(* IEC 61131-3 sources: Lasal/CPU_5344_V01/Class/switchesAxis, 1 file *)

(* ---- switchesAxis.st ---- *)
(*!
<Class
	Name               = "switchesAxis"
	Revision           = "0.0"
	RealtimeTask       = "false"
	CyclicTask         = "false"
	BackgroundTask     = "false"
	Sigmatek           = "false"
	OSInterface        = "false"
	HighPriority       = "false"
	Automatic          = "false"
	UpdateMode         = "Prescan"
	SharedCommandTable = "true"
	Objectsize         = "(284,120)">
	<Channels>
		<Server Name="ClassSvr" Visualized="false" Initialize="false" WriteProtected="true" Retentive="false"/>
		<Server Name="maxSwitch" Visualized="false" Initialize="false" WriteProtected="true" Retentive="false"/>
		<Server Name="minSwitch" Visualized="false" Initialize="false" WriteProtected="true" Retentive="false"/>
		<Server Name="overRuleMax" Visualized="false" Initialize="false" WriteProtected="false" Retentive="false"/>
		<Server Name="overRuleMin" Visualized="false" Initialize="false" WriteProtected="false" Retentive="false"/>
		<Server Name="overRuleRef" Visualized="false" Initialize="false" WriteProtected="false" Retentive="false"/>
		<Server Name="refSwitch" Visualized="false" Initialize="false" WriteProtected="true" Retentive="false"/>
		<Server Name="switchMaxIsNormallyOpen" Visualized="false" Initialize="false" WriteProtected="false" Retentive="File"/>
		<Server Name="switchMinIsNormallyOpen" Visualized="false" Initialize="false" WriteProtected="false" Retentive="File"/>
		<Client Name="ctrlServo" Required="true" Internal="false"/>
		<Client Name="iEsMaxSwitch" Required="false" Internal="false"/>
		<Client Name="iEsMinSwitch" Required="false" Internal="false"/>
		<Client Name="iEsRefSwitch" Required="false" Internal="false"/>
	</Channels>
</Class>
*)
switchesAxis : CLASS
  //Servers:
	ClassSvr 	: SvrChCmd_DINT;
	minSwitch 	: SvrCh_DINT;
	maxSwitch 	: SvrCh_DINT;
	refSwitch 	: SvrCh_DINT;
	switchMinIsNormallyOpen 	: SvrCh_DINT;
	switchMaxIsNormallyOpen 	: SvrCh_DINT;
	overRuleMin 	: SvrCh_DINT;
	overRuleMax 	: SvrCh_DINT;
	overRuleRef 	: SvrCh_DINT;
  //Clients:
	iEsMinSwitch 	: CltCh_DINT;
	iEsMaxSwitch 	: CltCh_DINT;
	iEsRefSwitch 	: CltCh_DINT;
	ctrlServo 	: CltChCmd_cmServo;
  //Variables:
  //Functions:

	FUNCTION VIRTUAL GLOBAL minSwitch::Read
		VAR_OUTPUT
			output (EAX) 	: DINT;
		END_VAR;

	FUNCTION VIRTUAL GLOBAL maxSwitch::Read
		VAR_OUTPUT
			output (EAX) 	: DINT;
		END_VAR;

	FUNCTION VIRTUAL GLOBAL refSwitch::Read
		VAR_OUTPUT
			output (EAX) 	: DINT;
		END_VAR;
  //Tables:
	FUNCTION @STD
		VAR_OUTPUT
			ret_code	: CONFSTATES;
		END_VAR;
	FUNCTION GLOBAL TAB @CT_;
END_CLASS;

#pragma usingLtd cmServo

// JdK 22-3-2022: switchesAxis, connect the endswitches to the axis, also handles the simulation states, goal is to make it less work to go to and from simulation

FUNCTION VIRTUAL GLOBAL switchesAxis::minSwitch::Read
	VAR_OUTPUT
		output (EAX) 	: DINT;
	END_VAR

  iEsMinSwitch:= iEsMinSwitch.Read();
  IF overRuleMin<> 0 THEN
   minSwitch:= overRuleMin>0;
  ELSIF ctrlServo.stsAllSimuActive THEN
    IF ctrlServo.parRefDirPositive= 0 THEN
      minSwitch:= ctrlServo.stsSimRef; //homing negative
    ELSE
      minSwitch:= 0;
    END_IF;
  ELSE
    IF switchMinIsNormallyOpen THEN
      minSwitch:= iEsMinSwitch;
    ELSE
      minSwitch:= iEsMinSwitch= 0; //invert signal
    END_IF;
  END_IF;

	output := minSwitch;

END_FUNCTION

FUNCTION VIRTUAL GLOBAL switchesAxis::maxSwitch::Read
	VAR_OUTPUT
		output (EAX) 	: DINT;
	END_VAR

  iEsMaxSwitch:= iEsMaxSwitch.Read();
  IF overRuleMax<> 0 THEN
    maxSwitch:= overRuleMax>0;
  ELSIF ctrlServo.stsAllSimuActive THEN
    IF ctrlServo.parRefDirPositive= 1 THEN
      maxSwitch:= ctrlServo.stsSimRef; //homing positive
    ELSE
      MaxSwitch:= 0;
    END_IF;
  ELSE
    IF switchMaxIsNormallyOpen THEN
      maxSwitch:= iEsMaxSwitch;
    ELSE
      maxSwitch:= iEsMaxSwitch= 0; //invert signal
    END_IF;
  END_IF;
	output := maxSwitch;

END_FUNCTION

FUNCTION VIRTUAL GLOBAL switchesAxis::refSwitch::Read
	VAR_OUTPUT
		output (EAX) 	: DINT;
	END_VAR

  iEsRefSwitch:= iEsRefSwitch.Read();
  IF overRuleRef<> 0 THEN
    refSwitch:= overRuleRef>0;
  ELSIF ctrlServo.stsAllSimuActive & ctrlServo.parNoRefSwitch= 0 THEN
    refSwitch:= ctrlServo.stsSimRef;
  ELSE
    refSwitch:= iEsRefSwitch;
  END_IF;

	output := refSwitch;

END_FUNCTION
